Universal Robots PolyScope program: Museum.urp

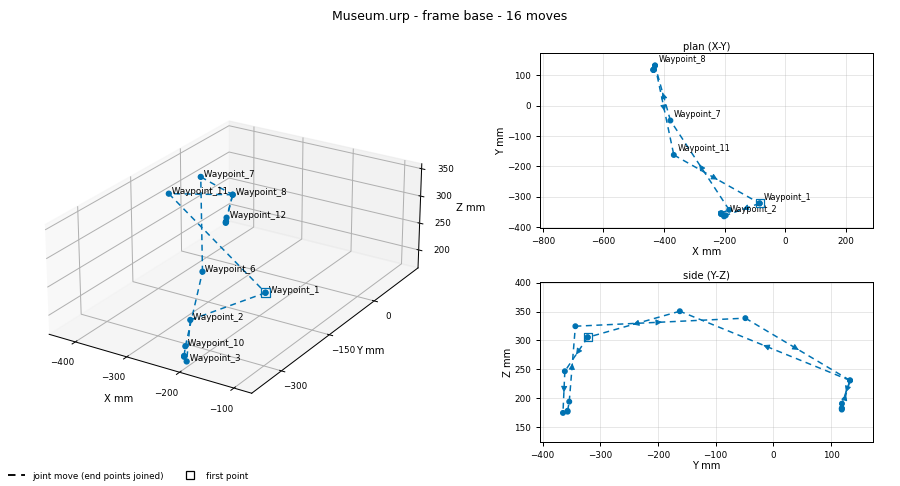
[picture p0: tool path of Museum.urp in frame base, 16 of 16 moves have a stored position in this frame; points joined in program order, loops and branches not executed]
Program Museum (installation=default directory=/programs/usbdisk/Zahra1 createdIn=5.11.11.1010533 lastSavedIn=5.11.11.1010533 robotSerialNumber=20205300864)
Calibrated DH parameters: a=[-0.000166, -0.243494, -0.153108, 0.000057, -0.000123, 0]; d=[0.151897, -1.34267, 53.988124, -52.514559, 0.085283, 0.092193]; alpha=[1.572472, -0.003756, 0.002824, 1.570807, -1.572621, 0]; deltaTheta=[0, 0.020704, 7.033215, -0.770746, 0.000004, 0]
Robot Program (runOnlyOnce=true)
  MoveJ speed 60 deg/s, acceleration 80 deg/s^2 (useActiveTCP=true) feature=Base
    Waypoint Waypoint_1: TCP in base x=-84.299 y=-321.875 z=305.481 mm, rx=-2.0809 ry=-2.2572 rz=0.0984 rad; joints [-79.978, -91.201, -87.971, -91.7, 84.671, 815.506] deg
    URCap Gripper Activate (Robotiq_Grippers, Robotiq Inc.) dataModel(ResetAndActivateKey=false)
    URCap Gripper (Robotiq_Grippers, Robotiq Inc.) dataModel(position=32.15686274509804, force=50.0, speed=18.0, positionInDouble=32.15686274509804, forceInDouble=50.0, speedInDouble=18.0, slaveIds=[9], blocking=true, robotCompliant=false)
    Waypoint Waypoint_2: TCP in base x=-196.445 y=-361.527 z=246.679 mm, rx=-3.1307 ry=-0.065 rz=0.1226 rad; joints [-98.988, -112.218, -78.42, -78.915, 85.468, 888.725] deg
    Waypoint Waypoint_3: TCP in base x=-201.975 y=-364.766 z=174.444 mm, rx=-3.1307 ry=-0.0651 rz=0.1226 rad; joints [-99.739, -119.118, -88.522, -61.858, 85.469, 887.999] deg
    Waypoint Waypoint_4: TCP in base x=-211.966 y=-356.714 z=176.563 mm, rx=3.1402 ry=0.0273 rz=0.003 rad; joints [-102.467, -119.007, -87.821, -63.021, 90.079, 886.679] deg
    URCap Gripper (Robotiq_Grippers, Robotiq Inc.) dataModel(position=83.15686274509804, force=73.0, speed=18.0, positionInDouble=83.15686274509804, forceInDouble=73.0, speedInDouble=18.0, slaveIds=[9], blocking=true, robotCompliant=false)
    Waypoint Waypoint_5: motionParameters(jointSpeed=0.698132 jointAcceleration=0.349066 cartesianSpeed=0.25 cartesianAcceleration=1.2); TCP in base x=-211.887 y=-356.801 z=178.071 mm, rx=3.1393 ry=0.0252 rz=0.0043 rad; joints [-102.466, -118.854, -87.634, -63.32, 90.137, 886.757] deg
    Waypoint Waypoint_10: TCP in base x=-211.313 y=-353.878 z=193.935 mm, rx=3.1146 ry=0.0248 rz=-0.0046 rad; joints [-102.472, -116.365, -87.526, -64.466, 90.138, 886.756] deg
    Waypoint Waypoint_6: TCP in base x=-185.149 y=-343.255 z=324.711 mm, rx=3.0545 ry=0.0796 rz=-0.0498 rad; joints [-98.543, -104.588, -69.726, -90.424, 88.968, 888.508] deg
    Waypoint Waypoint_7: TCP in base x=-378.997 y=-48.553 z=338.696 mm, rx=2.4027 ry=-1.9499 rz=-0.1309 rad; joints [-151.823, -102.958, -67.646, -95.069, 86.47, 916.243] deg
    Waypoint Waypoint_8: TCP in base x=-429.751 y=132.908 z=230.765 mm, rx=0.0068 ry=-3.0948 rz=0.012 rad; joints [-180.439, -122.61, -67.706, -76.903, 90.391, 989.41] deg
    Waypoint Waypoint_12: TCP in base x=-433.843 y=118.88 z=190.474 mm, rx=0.0081 ry=-3.1056 rz=-0.0549 rad; joints [-178.046, -125.089, -74.515, -68.323, 87.84, 991.724] deg
    Waypoint Waypoint_9: motionParameters(jointSpeed=0.698132 jointAcceleration=0.174533 cartesianSpeed=0.25 cartesianAcceleration=1.2); TCP in base x=-434.952 y=118.636 z=182.302 mm, rx=0.0089 ry=-3.1145 rz=-0.0543 rad; joints [-178.03, -126.142, -74.83, -67.465, 87.883, 991.726] deg
    Waypoint Waypoint_13: TCP in base x=-435.464 y=118.619 z=180.218 mm, rx=0.0091 ry=-3.117 rz=-0.0545 rad; joints [-178.03, -126.473, -74.795, -67.312, 87.882, 991.721] deg
    URCap Gripper (Robotiq_Grippers, Robotiq Inc.) dataModel(position=48.23529411764706, force=73.0, speed=18.0, positionInDouble=48.23529411764706, forceInDouble=73.0, speedInDouble=18.0, slaveIds=[9], blocking=true, robotCompliant=false)
    Waypoint Waypoint_9: motionParameters(jointSpeed=0.698132 jointAcceleration=0.174533 cartesianSpeed=0.25 cartesianAcceleration=1.2); TCP in base x=-434.952 y=118.636 z=182.302 mm, rx=0.0089 ry=-3.1145 rz=-0.0543 rad; joints [-178.03, -126.142, -74.83, -67.465, 87.883, 991.726] deg
    Waypoint Waypoint_8: TCP in base x=-429.751 y=132.908 z=230.765 mm, rx=0.0068 ry=-3.0948 rz=0.012 rad; joints [-180.439, -122.61, -67.706, -76.903, 90.391, 989.41] deg
    Waypoint Waypoint_11: TCP in base x=-367.743 y=-162.182 z=350.704 mm, rx=0.1181 ry=-3.0887 rz=-0.0197 rad; joints [-136.625, -110.695, -52.834, -104.666, 87.454, 1029.016] deg
    Waypoint Waypoint_1: TCP in base x=-84.299 y=-321.875 z=305.481 mm, rx=-2.0809 ry=-2.2572 rz=0.0984 rad; joints [-79.978, -91.201, -87.971, -91.7, 84.671, 815.506] deg
